Fanuc KAREL source: ka00205.KL

-- PROVISIONAL review KL for V940-1; original PC SHA256 43276284985672d442fa78b761f6ab3a60cfd51b5af5789d759c5f03543bab9d
-- Incomplete behavior may be omitted. Consult companion uncertainty JSON. Do not deploy.
PROGRAM KA00205
%NOLOCKGROUP
-- UNRESOLVED_DECL SRC type=002013
-- UNRESOLVED_DECL DST type=002013
BEGIN
  -- V9_COMPOSED_GLOBAL_TRANSFER_HINT repetitions=1; address IDs observed; pairing/direction/source/runtime held
  -- V9_TWO_GLOBAL_ADDRESS_COPY_HINT bounded five-record physical form; type/direction/source/runtime held
  -- V9_ZERO_TABLE_METADATA_HINT layout=0001; no indexed target words; source/name/runtime held
  -- UNRESOLVED_PC offsets 5-19; opcodes 22,22,1E
  -- UNRESOLVED_PC offsets 24-28; opcodes 7F
END KA00205
